FUNCTION_BLOCK FB_Roboter_E
VAR_INPUT
	bRefMax_in :BOOL;
	bRefMin_in :BOOL;
	
END_VAR
VAR_OUTPUT
	bRefMax_out :BOOL;
	bRefMin_out :BOOL;
	
END_VAR
VAR
END_VAR

bRefMax_out :=  NOT bRefMax_in;
bRefMin_out := NOT bRefMin_in;

END_FUNCTION_BLOCK

(* stored: Version 1.1.0.1, ProductVersion 3.1.4024.15
   POU FB_Roboter_E: Id {4af811a2-b766-4668-b73b-cadf1a937bf2}, SpecialFunc None *)
